FUNCTION_BLOCK ReworkDataManager EXTENDS TcoData.TcoDataExchange
VAR
    _data : ProcessData := (Parent := THIS^);
END_VAR

SUPER^();

PROPERTY Data : REFERENCE TO ProcessData
GET
Data REF= _data;
END_GET
END_PROPERTY

END_FUNCTION_BLOCK

(* stored: Version 1.1.0.1
   POU ReworkDataManager: Id {33b8f65c-34d7-4c88-b956-688f52621eeb}, SpecialFunc None
   Property Data: Id {98dcb715-feb5-4b56-9716-8495e81bdcc6}
   Get Get: Id {d372e65c-de3e-4aa8-b127-fd7616f5fc4b} *)
